TYPE CM_Motor_ALM :
STRUCT
END_STRUCT
END_TYPE

(* stored: Version 1.1.0.1, ProductVersion 3.1.4024.12
   DUT CM_Motor_ALM: Id {fa094ceb-4699-47cf-928f-7b6208f2d3de} *)
